// TIA Portal V17 export
// export: Created 2026-05-13T16:54:41.6864822Z, ExportSetting WithDefaults, DisplayName Totally Integrated Automation Portal, DisplayVersion V17 Update 4, DisplayName TIA Portal Openness, DisplayVersion V17 Update 4, DisplayName TIA Portal Version Control Interface, DisplayVersion V17, DisplayName SINAMICS Startdrive Advanced, DisplayVersion V17, DisplayName SINAMICS Startdrive G130, G150, S120, S150, SINAMICS MV, S210, DisplayVersion V17, DisplayName SINAMICS Startdrive G110M, G120, G120C, G120D, G120P, G115D, DisplayVersion V17, DisplayName STEP 7 Professional, DisplayVersion V17 Update 4, DisplayName STEP 7 Safety, DisplayVersion V17, DisplayName WinCC Professional, DisplayVersion V17 Update 4
TagTable "IOM"
  IYF引风机故障 : Bool  (PLC tag IYF引风机故障, HMI_连接_1, 100 ms)
  IDL电力调整器 : Bool  (PLC tag IDL电力调整器, HMI_连接_1, 100 ms)
  ILX离心雾化 : Bool  (PLC tag ILX离心雾化, HMI_连接_1, 100 ms)
  IJT急停 : Bool  (PLC tag IJT急停, HMI_连接_1, 100 ms)
  QDJ电加热 : Bool  (PLC tag QDJ电加热, HMI_连接_1, 100 ms)
  QYF引风机 : Bool  (PLC tag QYF引风机, HMI_连接_1, 100 ms)
  QLX离心雾化 : Bool  (PLC tag QLX离心雾化, HMI_连接_1, 100 ms)
  QJL进料泵 : Bool  (PLC tag QJL进料泵, HMI_连接_1, 100 ms)
  QJL进料泵正反 : Bool  (PLC tag QJL进料泵正反, HMI_连接_1, 100 ms)
  QHW恒温系统 : Bool  (PLC tag QHW恒温系统, HMI_连接_1, 100 ms)
  QZM照明 : Bool  (PLC tag QZM照明, HMI_连接_1, 100 ms)
  QRS热水炉 : Bool  (PLC tag QRS热水炉, HMI_连接_1, 100 ms)
  QBD布袋反吹1 : Bool  (PLC tag QBD布袋反吹1, HMI_连接_1, 100 ms)
  QBD布袋反吹2 : Bool  (PLC tag QBD布袋反吹2, HMI_连接_1, 100 ms)
  QBD布袋反吹3 : Bool  (PLC tag QBD布袋反吹3, HMI_连接_1, 100 ms)
  QZT主塔气扫1# : Bool  (PLC tag QZT主塔气扫1#, HMI_连接_1, 100 ms)
  QZT主塔气扫2# : Bool  (PLC tag QZT主塔气扫2#, HMI_连接_1, 100 ms)
  QZT主塔振打3# : Bool  (PLC tag QZT主塔振打3#, HMI_连接_1, 100 ms)
  QZT主塔气锤1# : Bool  (PLC tag QZT主塔气锤1#, HMI_连接_1, 100 ms)
  QZT主塔气锤2# : Bool  (PLC tag QZT主塔气锤2#, HMI_连接_1, 100 ms)
  QZT主塔气锤3# : Bool  (PLC tag QZT主塔气锤3#, HMI_连接_1, 100 ms)
  QQD气动锤备用1# : Bool  (PLC tag QQD气动锤备用1#, HMI_连接_1, 100 ms)
  QQD气动锤备用2# : Bool  (PLC tag QQD气动锤备用2#, HMI_连接_1, 100 ms)
  QQD气动锤备用3# : Bool  (PLC tag QQD气动锤备用3#, HMI_连接_1, 100 ms)
  QQD气动锤备用4# : Bool  (PLC tag QQD气动锤备用4#, HMI_连接_1, 100 ms)
  QBD布袋气锤1# : Bool  (PLC tag QBD布袋气锤1#, HMI_连接_1, 100 ms)
  QBD布袋气锤2# : Bool  (PLC tag QBD布袋气锤2#, HMI_连接_1, 100 ms)
  QBD布袋气锤3# : Bool  (PLC tag QBD布袋气锤3#, HMI_连接_1, 100 ms)
  QFM蜂鸣器 : Bool  (PLC tag QFM蜂鸣器, HMI_连接_1, 100 ms)
